(* Logix 5000 project; controller AMANA_DC_PLANT_01 vendor 1 type 14 code 164 rev 31.12; software revision 31.02; part 8 of 9 *)
(* tags used below, declared in another part *)
   Barcode_Longest : DINT;
   Barcode_Shortest : DINT;
   Comma : STRING;
   NULL_String : STRING;
   SCANNER_LN467MERGE_DATA : Keyence_2_Barcode;
   SCANNER_LONGTERMEAST_DATA : Keyence_2_Barcode;
   SCANNER_LONGTERMWEST_DATA : Keyence_2_Barcode;
   SCANNER_WAREHOUSENORTH_DATA : Keyence_2_Barcode;
   SCANNER_WAREHOUSESOUTH_DATA : Keyence_2_Barcode;
(* OH_BARCODE_SCAN, continued *)

ROUTINE R06_WAREHOUSENORTH   (* ladder *)
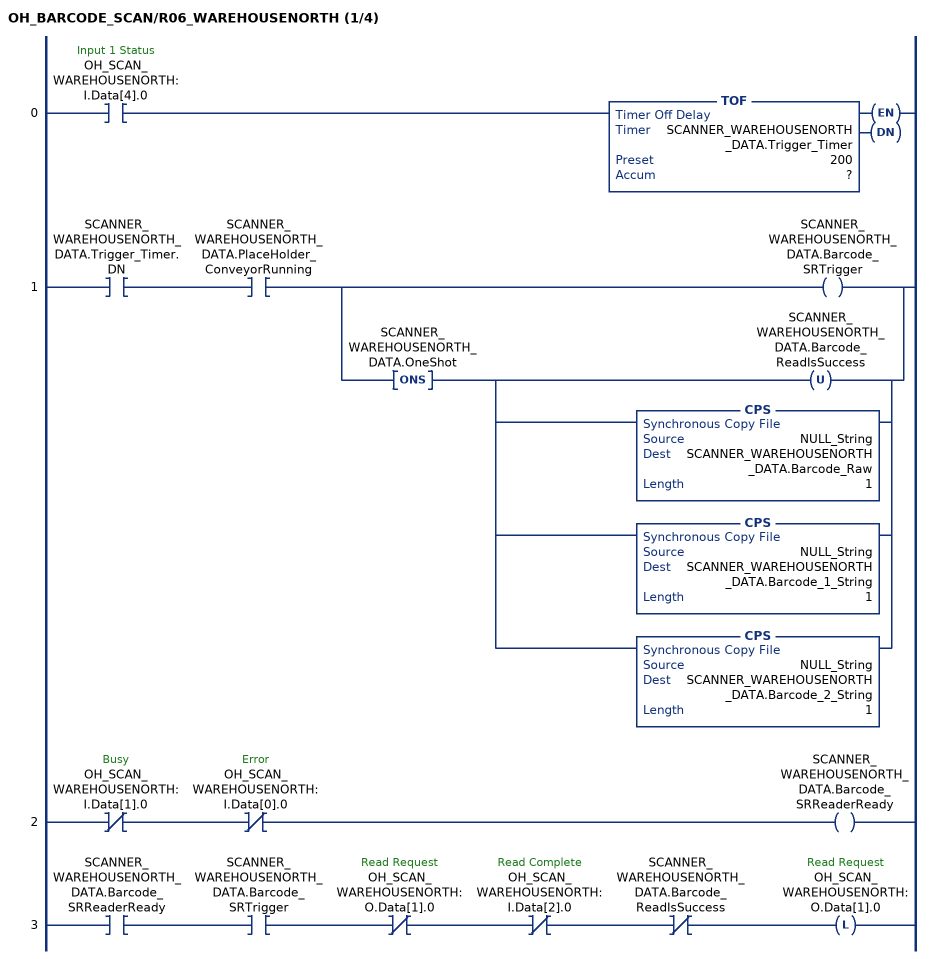
   0: XIC(OH_SCAN_WAREHOUSENORTH:I.Data[4].0)TOF(SCANNER_WAREHOUSENORTH_DATA.Trigger_Timer,?,?);
   1: XIC(SCANNER_WAREHOUSENORTH_DATA.Trigger_Timer.DN)XIC(SCANNER_WAREHOUSENORTH_DATA.PlaceHolder_ConveyorRunning)[OTE(SCANNER_WAREHOUSENORTH_DATA.Barcode_SRTrigger) ,ONS(SCANNER_WAREHOUSENORTH_DATA.OneShot) [OTU(SCANNER_WAREHOUSENORTH_DATA.Barcode_ReadIsSuccess) ,CPS(NULL_String,SCANNER_WAREHOUSENORTH_DATA.Barcode_Raw,1) ,CPS(NULL_String,SCANNER_WAREHOUSENORTH_DATA.Barcode_1_String,1) ,CPS(NULL_String,SCANNER_WAREHOUSENORTH_DATA.Barcode_2_String,1) ] ];
   2: XIO(OH_SCAN_WAREHOUSENORTH:I.Data[1].0)XIO(OH_SCAN_WAREHOUSENORTH:I.Data[0].0)OTE(SCANNER_WAREHOUSENORTH_DATA.Barcode_SRReaderReady);
   3: XIC(SCANNER_WAREHOUSENORTH_DATA.Barcode_SRReaderReady)XIC(SCANNER_WAREHOUSENORTH_DATA.Barcode_SRTrigger)XIO(OH_SCAN_WAREHOUSENORTH:O.Data[1].0)XIO(OH_SCAN_WAREHOUSENORTH:I.Data[2].0)XIO(SCANNER_WAREHOUSENORTH_DATA.Barcode_ReadIsSuccess)OTL(OH_SCAN_WAREHOUSENORTH:O.Data[1].0);
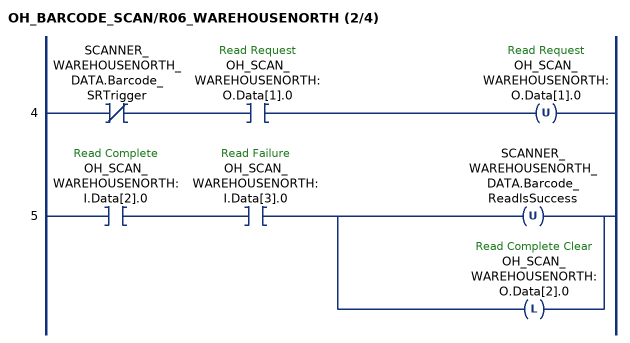
   4: XIO(SCANNER_WAREHOUSENORTH_DATA.Barcode_SRTrigger)XIC(OH_SCAN_WAREHOUSENORTH:O.Data[1].0)OTU(OH_SCAN_WAREHOUSENORTH:O.Data[1].0);
   5: XIC(OH_SCAN_WAREHOUSENORTH:I.Data[2].0)XIC(OH_SCAN_WAREHOUSENORTH:I.Data[3].0)[OTU(SCANNER_WAREHOUSENORTH_DATA.Barcode_ReadIsSuccess) ,OTL(OH_SCAN_WAREHOUSENORTH:O.Data[2].0) ];
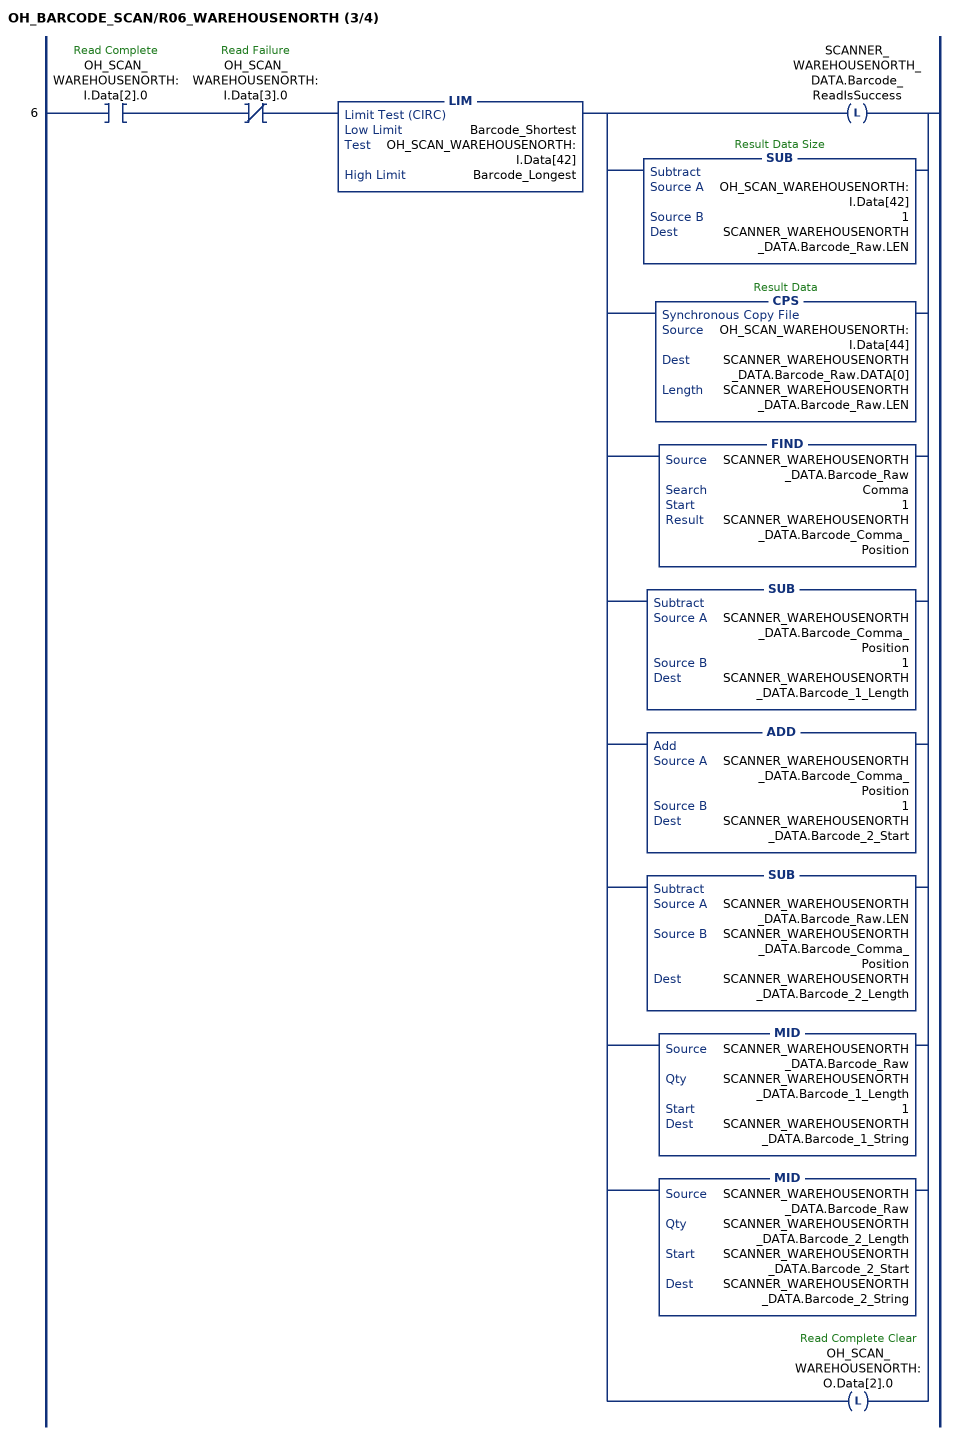
   6: XIC(OH_SCAN_WAREHOUSENORTH:I.Data[2].0)XIO(OH_SCAN_WAREHOUSENORTH:I.Data[3].0)LIM(Barcode_Shortest,OH_SCAN_WAREHOUSENORTH:I.Data[42],Barcode_Longest)[OTL(SCANNER_WAREHOUSENORTH_DATA.Barcode_ReadIsSuccess) ,SUB(OH_SCAN_WAREHOUSENORTH:I.Data[42],1,SCANNER_WAREHOUSENORTH_DATA.Barcode_Raw.LEN) ,CPS(OH_SCAN_WAREHOUSENORTH:I.Data[44],SCANNER_WAREHOUSENORTH_DATA.Barcode_Raw.DATA[0],SCANNER_WAREHOUSENORTH_DATA.Barcode_Raw.LEN) ,FIND(SCANNER_WAREHOUSENORTH_DATA.Barcode_Raw,Comma,1,SCANNER_WAREHOUSENORTH_DATA.Barcode_Comma_Position) ,SUB(SCANNER_WAREHOUSENORTH_DATA.Barcode_Comma_Position,1,SCANNER_WAREHOUSENORTH_DATA.Barcode_1_Length) ,ADD(SCANNER_WAREHOUSENORTH_DATA.Barcode_Comma_Position,1,SCANNER_WAREHOUSENORTH_DATA.Barcode_2_Start) ,SUB(SCANNER_WAREHOUSENORTH_DATA.Barcode_Raw.LEN,SCANNER_WAREHOUSENORTH_DATA.Barcode_Comma_Position,SCANNER_WAREHOUSENORTH_DATA.Barcode_2_Length) ,MID(SCANNER_WAREHOUSENORTH_DATA.Barcode_Raw,SCANNER_WAREHOUSENORTH_DATA.Barcode_1_Length,1,SCANNER_WAREHOUSENORTH_DATA.Barcode_1_String) ,MID(SCANNER_WAREHOUSENORTH_DATA.Barcode_Raw,SCANNER_WAREHOUSENORTH_DATA.Barcode_2_Length,SCANNER_WAREHOUSENORTH_DATA.Barcode_2_Start,SCANNER_WAREHOUSENORTH_DATA.Barcode_2_String) ,OTL(OH_SCAN_WAREHOUSENORTH:O.Data[2].0) ];
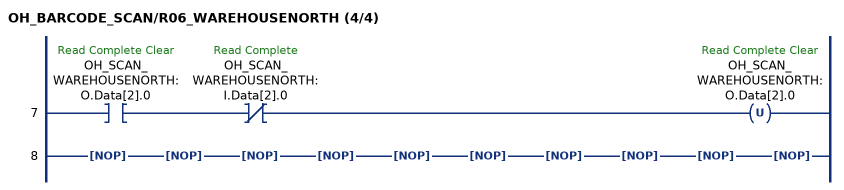
   7: XIC(OH_SCAN_WAREHOUSENORTH:O.Data[2].0)XIO(OH_SCAN_WAREHOUSENORTH:I.Data[2].0)OTU(OH_SCAN_WAREHOUSENORTH:O.Data[2].0);
   8: NOP()NOP()NOP()NOP()NOP()NOP()NOP()NOP()NOP()NOP();
END_ROUTINE

ROUTINE R07_WAREHOUSESOUTH   (* ladder *)
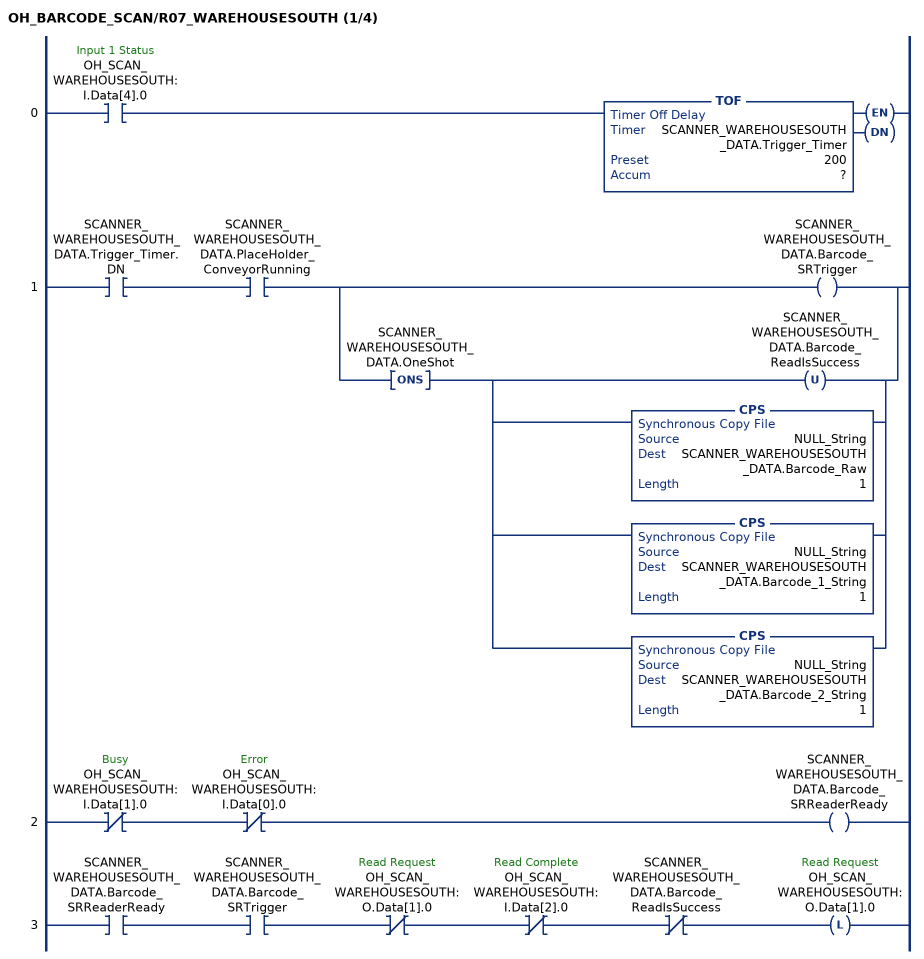
   0: XIC(OH_SCAN_WAREHOUSESOUTH:I.Data[4].0)TOF(SCANNER_WAREHOUSESOUTH_DATA.Trigger_Timer,?,?);
   1: XIC(SCANNER_WAREHOUSESOUTH_DATA.Trigger_Timer.DN)XIC(SCANNER_WAREHOUSESOUTH_DATA.PlaceHolder_ConveyorRunning)[OTE(SCANNER_WAREHOUSESOUTH_DATA.Barcode_SRTrigger) ,ONS(SCANNER_WAREHOUSESOUTH_DATA.OneShot) [OTU(SCANNER_WAREHOUSESOUTH_DATA.Barcode_ReadIsSuccess) ,CPS(NULL_String,SCANNER_WAREHOUSESOUTH_DATA.Barcode_Raw,1) ,CPS(NULL_String,SCANNER_WAREHOUSESOUTH_DATA.Barcode_1_String,1) ,CPS(NULL_String,SCANNER_WAREHOUSESOUTH_DATA.Barcode_2_String,1) ] ];
   2: XIO(OH_SCAN_WAREHOUSESOUTH:I.Data[1].0)XIO(OH_SCAN_WAREHOUSESOUTH:I.Data[0].0)OTE(SCANNER_WAREHOUSESOUTH_DATA.Barcode_SRReaderReady);
   3: XIC(SCANNER_WAREHOUSESOUTH_DATA.Barcode_SRReaderReady)XIC(SCANNER_WAREHOUSESOUTH_DATA.Barcode_SRTrigger)XIO(OH_SCAN_WAREHOUSESOUTH:O.Data[1].0)XIO(OH_SCAN_WAREHOUSESOUTH:I.Data[2].0)XIO(SCANNER_WAREHOUSESOUTH_DATA.Barcode_ReadIsSuccess)OTL(OH_SCAN_WAREHOUSESOUTH:O.Data[1].0);
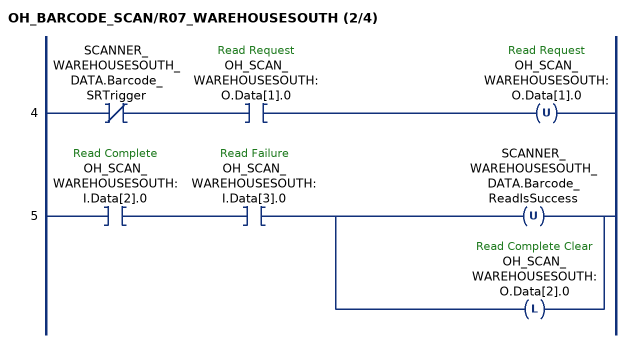
   4: XIO(SCANNER_WAREHOUSESOUTH_DATA.Barcode_SRTrigger)XIC(OH_SCAN_WAREHOUSESOUTH:O.Data[1].0)OTU(OH_SCAN_WAREHOUSESOUTH:O.Data[1].0);
   5: XIC(OH_SCAN_WAREHOUSESOUTH:I.Data[2].0)XIC(OH_SCAN_WAREHOUSESOUTH:I.Data[3].0)[OTU(SCANNER_WAREHOUSESOUTH_DATA.Barcode_ReadIsSuccess) ,OTL(OH_SCAN_WAREHOUSESOUTH:O.Data[2].0) ];
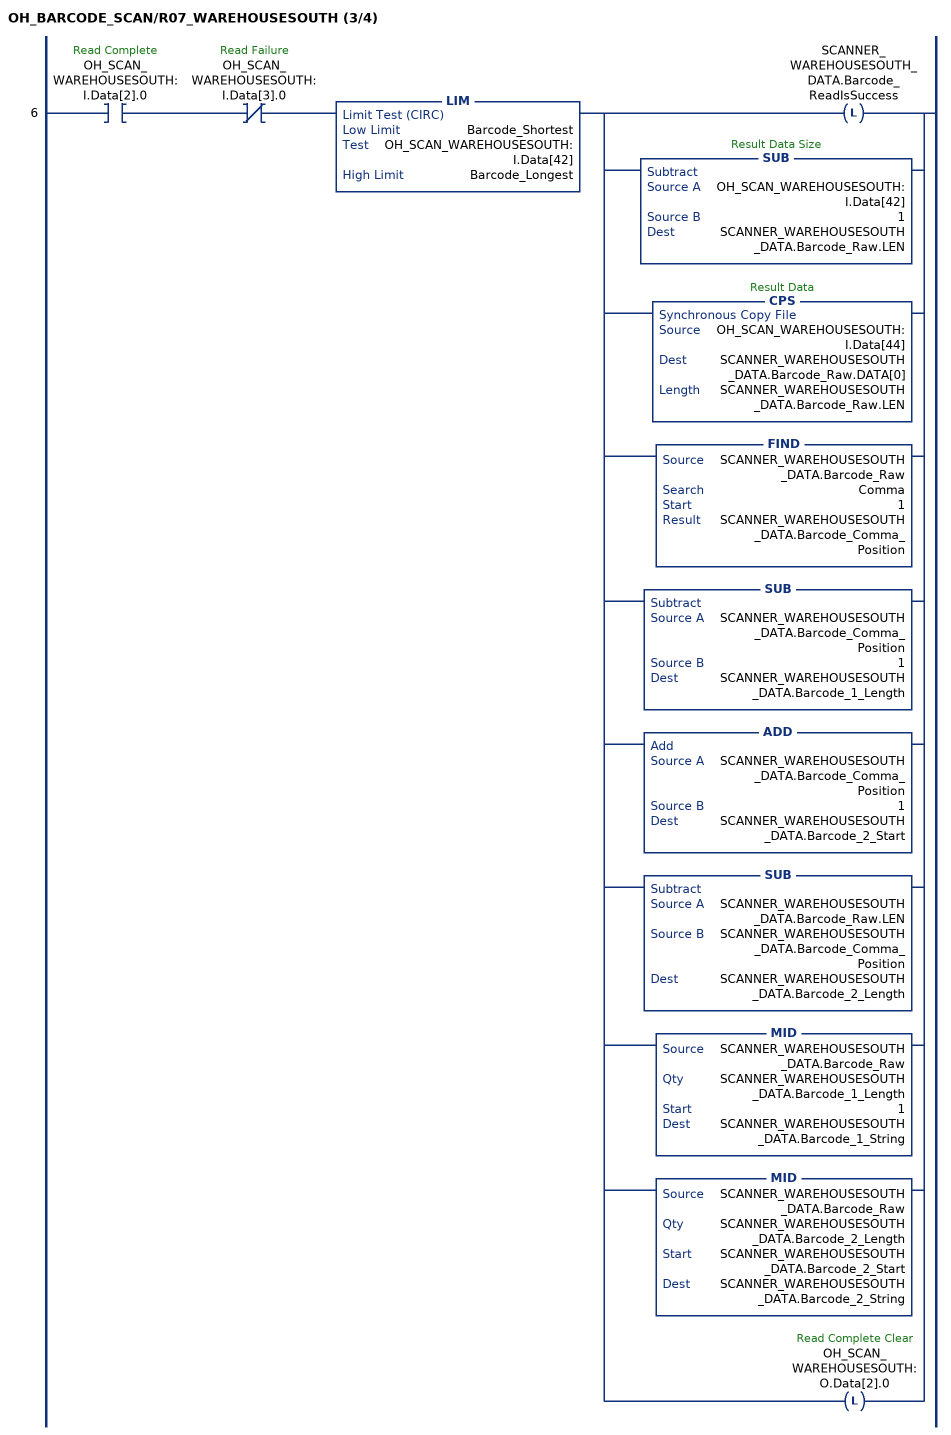
   6: XIC(OH_SCAN_WAREHOUSESOUTH:I.Data[2].0)XIO(OH_SCAN_WAREHOUSESOUTH:I.Data[3].0)LIM(Barcode_Shortest,OH_SCAN_WAREHOUSESOUTH:I.Data[42],Barcode_Longest)[OTL(SCANNER_WAREHOUSESOUTH_DATA.Barcode_ReadIsSuccess) ,SUB(OH_SCAN_WAREHOUSESOUTH:I.Data[42],1,SCANNER_WAREHOUSESOUTH_DATA.Barcode_Raw.LEN) ,CPS(OH_SCAN_WAREHOUSESOUTH:I.Data[44],SCANNER_WAREHOUSESOUTH_DATA.Barcode_Raw.DATA[0],SCANNER_WAREHOUSESOUTH_DATA.Barcode_Raw.LEN) ,FIND(SCANNER_WAREHOUSESOUTH_DATA.Barcode_Raw,Comma,1,SCANNER_WAREHOUSESOUTH_DATA.Barcode_Comma_Position) ,SUB(SCANNER_WAREHOUSESOUTH_DATA.Barcode_Comma_Position,1,SCANNER_WAREHOUSESOUTH_DATA.Barcode_1_Length) ,ADD(SCANNER_WAREHOUSESOUTH_DATA.Barcode_Comma_Position,1,SCANNER_WAREHOUSESOUTH_DATA.Barcode_2_Start) ,SUB(SCANNER_WAREHOUSESOUTH_DATA.Barcode_Raw.LEN,SCANNER_WAREHOUSESOUTH_DATA.Barcode_Comma_Position,SCANNER_WAREHOUSESOUTH_DATA.Barcode_2_Length) ,MID(SCANNER_WAREHOUSESOUTH_DATA.Barcode_Raw,SCANNER_WAREHOUSESOUTH_DATA.Barcode_1_Length,1,SCANNER_WAREHOUSESOUTH_DATA.Barcode_1_String) ,MID(SCANNER_WAREHOUSESOUTH_DATA.Barcode_Raw,SCANNER_WAREHOUSESOUTH_DATA.Barcode_2_Length,SCANNER_WAREHOUSESOUTH_DATA.Barcode_2_Start,SCANNER_WAREHOUSESOUTH_DATA.Barcode_2_String) ,OTL(OH_SCAN_WAREHOUSESOUTH:O.Data[2].0) ];
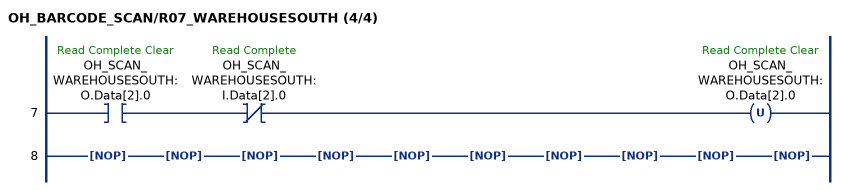
   7: XIC(OH_SCAN_WAREHOUSESOUTH:O.Data[2].0)XIO(OH_SCAN_WAREHOUSESOUTH:I.Data[2].0)OTU(OH_SCAN_WAREHOUSESOUTH:O.Data[2].0);
   8: NOP()NOP()NOP()NOP()NOP()NOP()NOP()NOP()NOP()NOP();
END_ROUTINE

ROUTINE R08_LONGTERMEAST   (* ladder *)
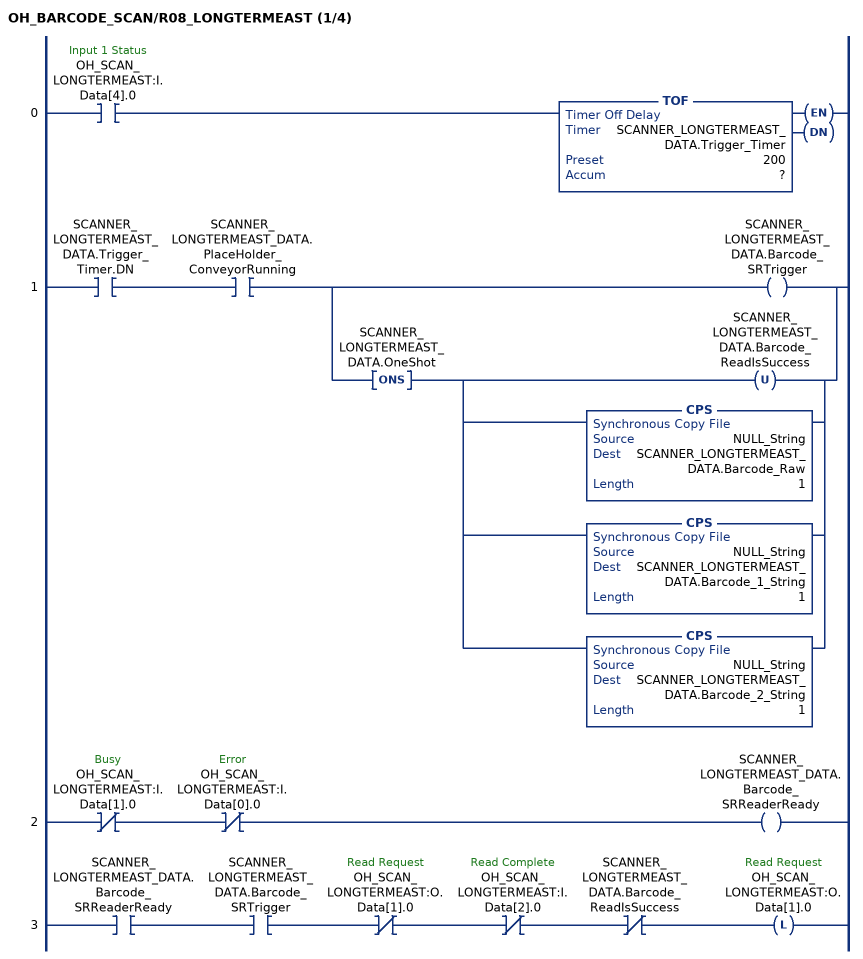
   0: XIC(OH_SCAN_LONGTERMEAST:I.Data[4].0)TOF(SCANNER_LONGTERMEAST_DATA.Trigger_Timer,?,?);
   1: XIC(SCANNER_LONGTERMEAST_DATA.Trigger_Timer.DN)XIC(SCANNER_LONGTERMEAST_DATA.PlaceHolder_ConveyorRunning)[OTE(SCANNER_LONGTERMEAST_DATA.Barcode_SRTrigger) ,ONS(SCANNER_LONGTERMEAST_DATA.OneShot) [OTU(SCANNER_LONGTERMEAST_DATA.Barcode_ReadIsSuccess) ,CPS(NULL_String,SCANNER_LONGTERMEAST_DATA.Barcode_Raw,1) ,CPS(NULL_String,SCANNER_LONGTERMEAST_DATA.Barcode_1_String,1) ,CPS(NULL_String,SCANNER_LONGTERMEAST_DATA.Barcode_2_String,1) ] ];
   2: XIO(OH_SCAN_LONGTERMEAST:I.Data[1].0)XIO(OH_SCAN_LONGTERMEAST:I.Data[0].0)OTE(SCANNER_LONGTERMEAST_DATA.Barcode_SRReaderReady);
   3: XIC(SCANNER_LONGTERMEAST_DATA.Barcode_SRReaderReady)XIC(SCANNER_LONGTERMEAST_DATA.Barcode_SRTrigger)XIO(OH_SCAN_LONGTERMEAST:O.Data[1].0)XIO(OH_SCAN_LONGTERMEAST:I.Data[2].0)XIO(SCANNER_LONGTERMEAST_DATA.Barcode_ReadIsSuccess)OTL(OH_SCAN_LONGTERMEAST:O.Data[1].0);
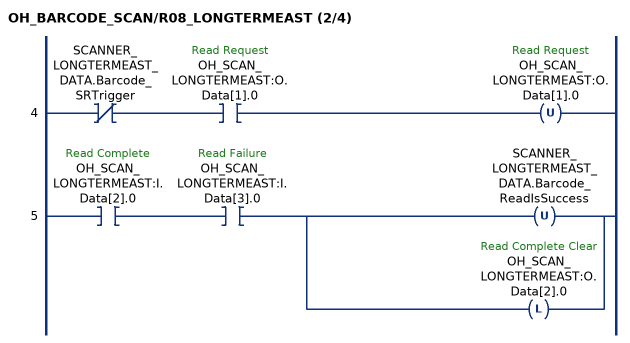
   4: XIO(SCANNER_LONGTERMEAST_DATA.Barcode_SRTrigger)XIC(OH_SCAN_LONGTERMEAST:O.Data[1].0)OTU(OH_SCAN_LONGTERMEAST:O.Data[1].0);
   5: XIC(OH_SCAN_LONGTERMEAST:I.Data[2].0)XIC(OH_SCAN_LONGTERMEAST:I.Data[3].0)[OTU(SCANNER_LONGTERMEAST_DATA.Barcode_ReadIsSuccess) ,OTL(OH_SCAN_LONGTERMEAST:O.Data[2].0) ];
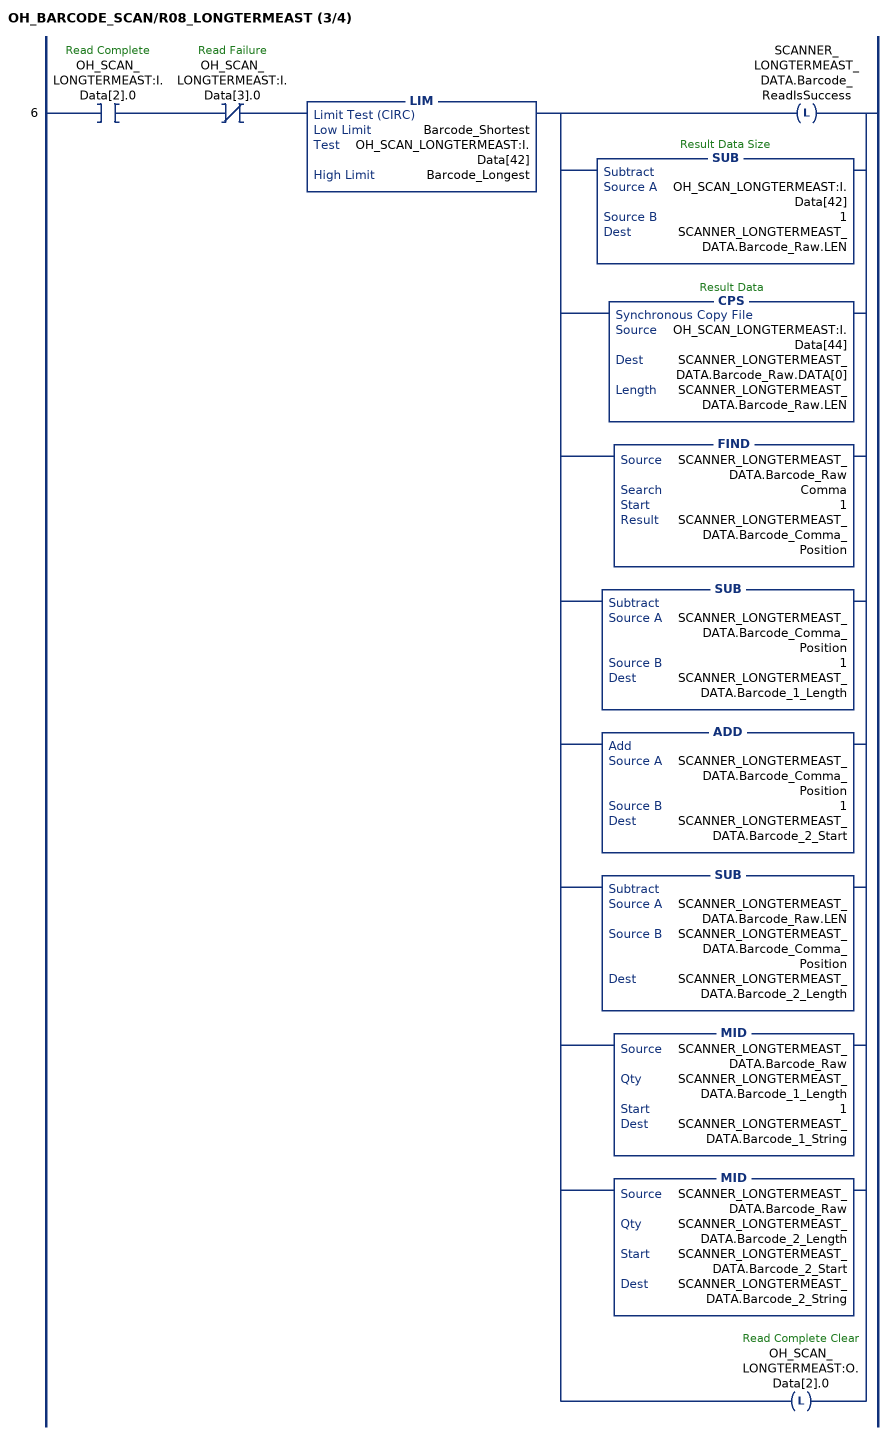
   6: XIC(OH_SCAN_LONGTERMEAST:I.Data[2].0)XIO(OH_SCAN_LONGTERMEAST:I.Data[3].0)LIM(Barcode_Shortest,OH_SCAN_LONGTERMEAST:I.Data[42],Barcode_Longest)[OTL(SCANNER_LONGTERMEAST_DATA.Barcode_ReadIsSuccess) ,SUB(OH_SCAN_LONGTERMEAST:I.Data[42],1,SCANNER_LONGTERMEAST_DATA.Barcode_Raw.LEN) ,CPS(OH_SCAN_LONGTERMEAST:I.Data[44],SCANNER_LONGTERMEAST_DATA.Barcode_Raw.DATA[0],SCANNER_LONGTERMEAST_DATA.Barcode_Raw.LEN) ,FIND(SCANNER_LONGTERMEAST_DATA.Barcode_Raw,Comma,1,SCANNER_LONGTERMEAST_DATA.Barcode_Comma_Position) ,SUB(SCANNER_LONGTERMEAST_DATA.Barcode_Comma_Position,1,SCANNER_LONGTERMEAST_DATA.Barcode_1_Length) ,ADD(SCANNER_LONGTERMEAST_DATA.Barcode_Comma_Position,1,SCANNER_LONGTERMEAST_DATA.Barcode_2_Start) ,SUB(SCANNER_LONGTERMEAST_DATA.Barcode_Raw.LEN,SCANNER_LONGTERMEAST_DATA.Barcode_Comma_Position,SCANNER_LONGTERMEAST_DATA.Barcode_2_Length) ,MID(SCANNER_LONGTERMEAST_DATA.Barcode_Raw,SCANNER_LONGTERMEAST_DATA.Barcode_1_Length,1,SCANNER_LONGTERMEAST_DATA.Barcode_1_String) ,MID(SCANNER_LONGTERMEAST_DATA.Barcode_Raw,SCANNER_LONGTERMEAST_DATA.Barcode_2_Length,SCANNER_LONGTERMEAST_DATA.Barcode_2_Start,SCANNER_LONGTERMEAST_DATA.Barcode_2_String) ,OTL(OH_SCAN_LONGTERMEAST:O.Data[2].0) ];
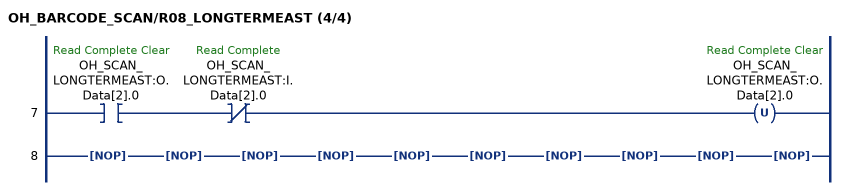
   7: XIC(OH_SCAN_LONGTERMEAST:O.Data[2].0)XIO(OH_SCAN_LONGTERMEAST:I.Data[2].0)OTU(OH_SCAN_LONGTERMEAST:O.Data[2].0);
   8: NOP()NOP()NOP()NOP()NOP()NOP()NOP()NOP()NOP()NOP();
END_ROUTINE

ROUTINE R09_LONGTERMWEST   (* ladder *)
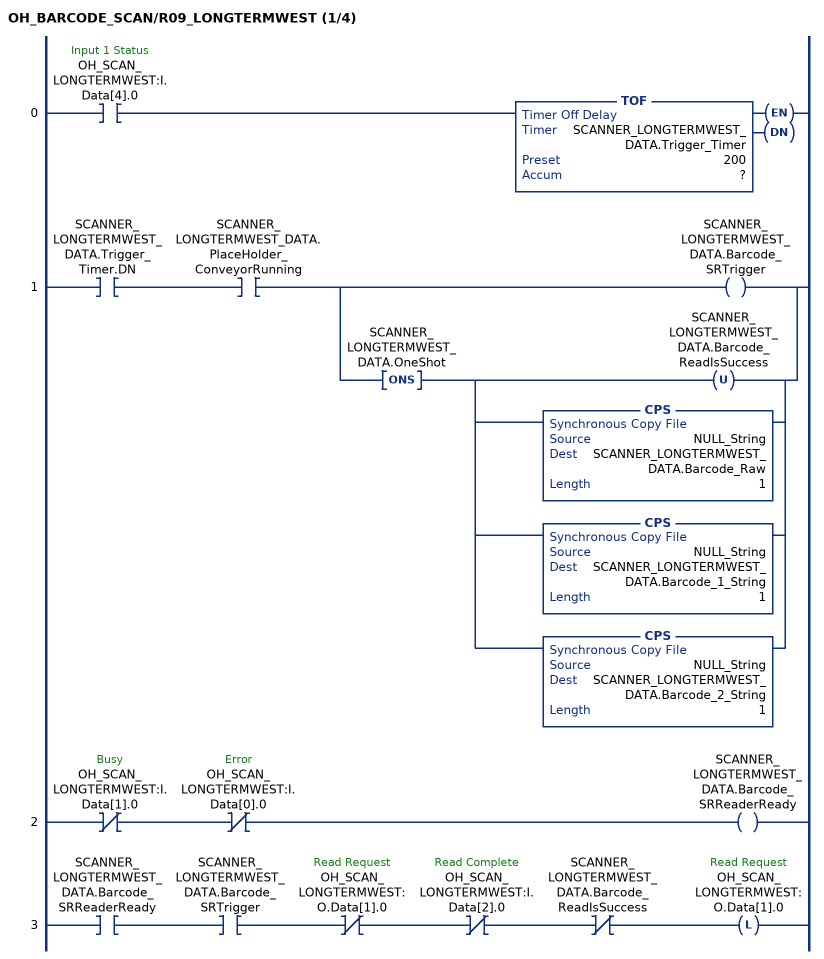
   0: XIC(OH_SCAN_LONGTERMWEST:I.Data[4].0)TOF(SCANNER_LONGTERMWEST_DATA.Trigger_Timer,?,?);
   1: XIC(SCANNER_LONGTERMWEST_DATA.Trigger_Timer.DN)XIC(SCANNER_LONGTERMWEST_DATA.PlaceHolder_ConveyorRunning)[OTE(SCANNER_LONGTERMWEST_DATA.Barcode_SRTrigger) ,ONS(SCANNER_LONGTERMWEST_DATA.OneShot) [OTU(SCANNER_LONGTERMWEST_DATA.Barcode_ReadIsSuccess) ,CPS(NULL_String,SCANNER_LONGTERMWEST_DATA.Barcode_Raw,1) ,CPS(NULL_String,SCANNER_LONGTERMWEST_DATA.Barcode_1_String,1) ,CPS(NULL_String,SCANNER_LONGTERMWEST_DATA.Barcode_2_String,1) ] ];
   2: XIO(OH_SCAN_LONGTERMWEST:I.Data[1].0)XIO(OH_SCAN_LONGTERMWEST:I.Data[0].0)OTE(SCANNER_LONGTERMWEST_DATA.Barcode_SRReaderReady);
   3: XIC(SCANNER_LONGTERMWEST_DATA.Barcode_SRReaderReady)XIC(SCANNER_LONGTERMWEST_DATA.Barcode_SRTrigger)XIO(OH_SCAN_LONGTERMWEST:O.Data[1].0)XIO(OH_SCAN_LONGTERMWEST:I.Data[2].0)XIO(SCANNER_LONGTERMWEST_DATA.Barcode_ReadIsSuccess)OTL(OH_SCAN_LONGTERMWEST:O.Data[1].0);
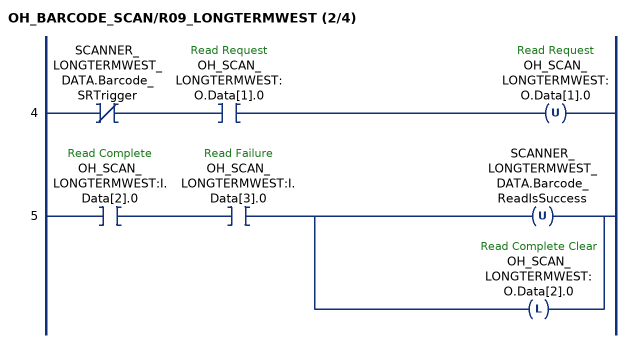
   4: XIO(SCANNER_LONGTERMWEST_DATA.Barcode_SRTrigger)XIC(OH_SCAN_LONGTERMWEST:O.Data[1].0)OTU(OH_SCAN_LONGTERMWEST:O.Data[1].0);
   5: XIC(OH_SCAN_LONGTERMWEST:I.Data[2].0)XIC(OH_SCAN_LONGTERMWEST:I.Data[3].0)[OTU(SCANNER_LONGTERMWEST_DATA.Barcode_ReadIsSuccess) ,OTL(OH_SCAN_LONGTERMWEST:O.Data[2].0) ];
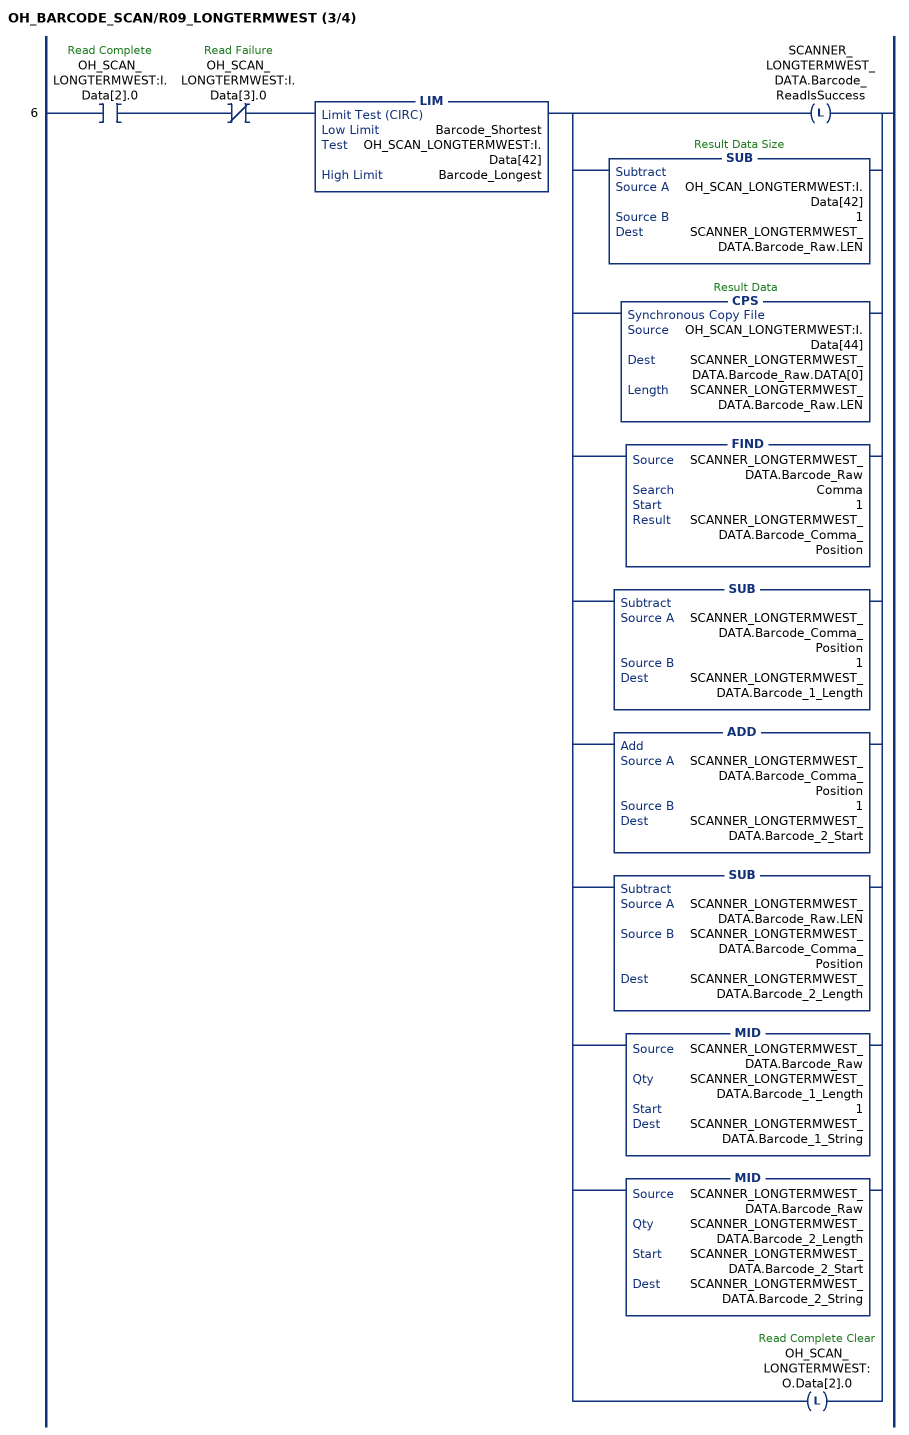
   6: XIC(OH_SCAN_LONGTERMWEST:I.Data[2].0)XIO(OH_SCAN_LONGTERMWEST:I.Data[3].0)LIM(Barcode_Shortest,OH_SCAN_LONGTERMWEST:I.Data[42],Barcode_Longest)[OTL(SCANNER_LONGTERMWEST_DATA.Barcode_ReadIsSuccess) ,SUB(OH_SCAN_LONGTERMWEST:I.Data[42],1,SCANNER_LONGTERMWEST_DATA.Barcode_Raw.LEN) ,CPS(OH_SCAN_LONGTERMWEST:I.Data[44],SCANNER_LONGTERMWEST_DATA.Barcode_Raw.DATA[0],SCANNER_LONGTERMWEST_DATA.Barcode_Raw.LEN) ,FIND(SCANNER_LONGTERMWEST_DATA.Barcode_Raw,Comma,1,SCANNER_LONGTERMWEST_DATA.Barcode_Comma_Position) ,SUB(SCANNER_LONGTERMWEST_DATA.Barcode_Comma_Position,1,SCANNER_LONGTERMWEST_DATA.Barcode_1_Length) ,ADD(SCANNER_LONGTERMWEST_DATA.Barcode_Comma_Position,1,SCANNER_LONGTERMWEST_DATA.Barcode_2_Start) ,SUB(SCANNER_LONGTERMWEST_DATA.Barcode_Raw.LEN,SCANNER_LONGTERMWEST_DATA.Barcode_Comma_Position,SCANNER_LONGTERMWEST_DATA.Barcode_2_Length) ,MID(SCANNER_LONGTERMWEST_DATA.Barcode_Raw,SCANNER_LONGTERMWEST_DATA.Barcode_1_Length,1,SCANNER_LONGTERMWEST_DATA.Barcode_1_String) ,MID(SCANNER_LONGTERMWEST_DATA.Barcode_Raw,SCANNER_LONGTERMWEST_DATA.Barcode_2_Length,SCANNER_LONGTERMWEST_DATA.Barcode_2_Start,SCANNER_LONGTERMWEST_DATA.Barcode_2_String) ,OTL(OH_SCAN_LONGTERMWEST:O.Data[2].0) ];
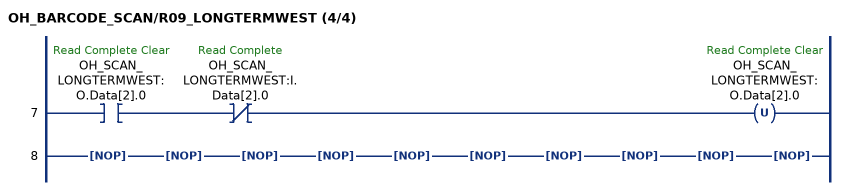
   7: XIC(OH_SCAN_LONGTERMWEST:O.Data[2].0)XIO(OH_SCAN_LONGTERMWEST:I.Data[2].0)OTU(OH_SCAN_LONGTERMWEST:O.Data[2].0);
   8: NOP()NOP()NOP()NOP()NOP()NOP()NOP()NOP()NOP()NOP();
END_ROUTINE

ROUTINE R10_LN467MERGE   (* ladder *)
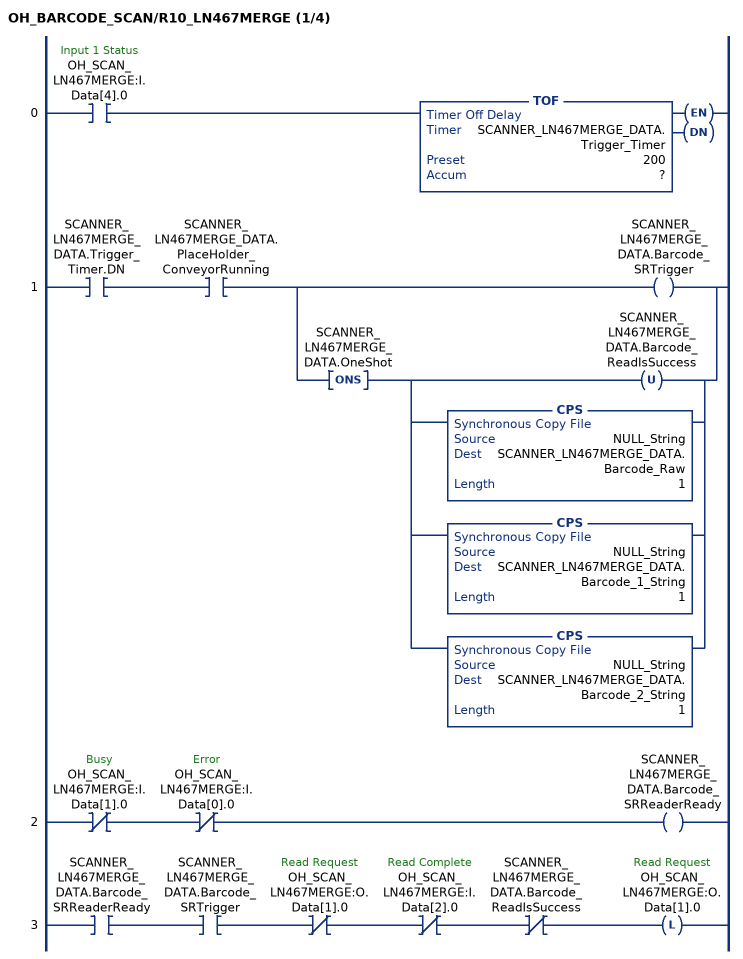
   0: XIC(OH_SCAN_LN467MERGE:I.Data[4].0)TOF(SCANNER_LN467MERGE_DATA.Trigger_Timer,?,?);
   1: XIC(SCANNER_LN467MERGE_DATA.Trigger_Timer.DN)XIC(SCANNER_LN467MERGE_DATA.PlaceHolder_ConveyorRunning)[OTE(SCANNER_LN467MERGE_DATA.Barcode_SRTrigger) ,ONS(SCANNER_LN467MERGE_DATA.OneShot) [OTU(SCANNER_LN467MERGE_DATA.Barcode_ReadIsSuccess) ,CPS(NULL_String,SCANNER_LN467MERGE_DATA.Barcode_Raw,1) ,CPS(NULL_String,SCANNER_LN467MERGE_DATA.Barcode_1_String,1) ,CPS(NULL_String,SCANNER_LN467MERGE_DATA.Barcode_2_String,1) ] ];
   2: XIO(OH_SCAN_LN467MERGE:I.Data[1].0)XIO(OH_SCAN_LN467MERGE:I.Data[0].0)OTE(SCANNER_LN467MERGE_DATA.Barcode_SRReaderReady);
   3: XIC(SCANNER_LN467MERGE_DATA.Barcode_SRReaderReady)XIC(SCANNER_LN467MERGE_DATA.Barcode_SRTrigger)XIO(OH_SCAN_LN467MERGE:O.Data[1].0)XIO(OH_SCAN_LN467MERGE:I.Data[2].0)XIO(SCANNER_LN467MERGE_DATA.Barcode_ReadIsSuccess)OTL(OH_SCAN_LN467MERGE:O.Data[1].0);
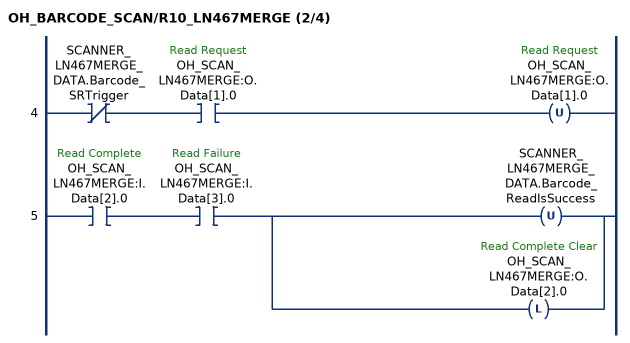
   4: XIO(SCANNER_LN467MERGE_DATA.Barcode_SRTrigger)XIC(OH_SCAN_LN467MERGE:O.Data[1].0)OTU(OH_SCAN_LN467MERGE:O.Data[1].0);
   5: XIC(OH_SCAN_LN467MERGE:I.Data[2].0)XIC(OH_SCAN_LN467MERGE:I.Data[3].0)[OTU(SCANNER_LN467MERGE_DATA.Barcode_ReadIsSuccess) ,OTL(OH_SCAN_LN467MERGE:O.Data[2].0) ];
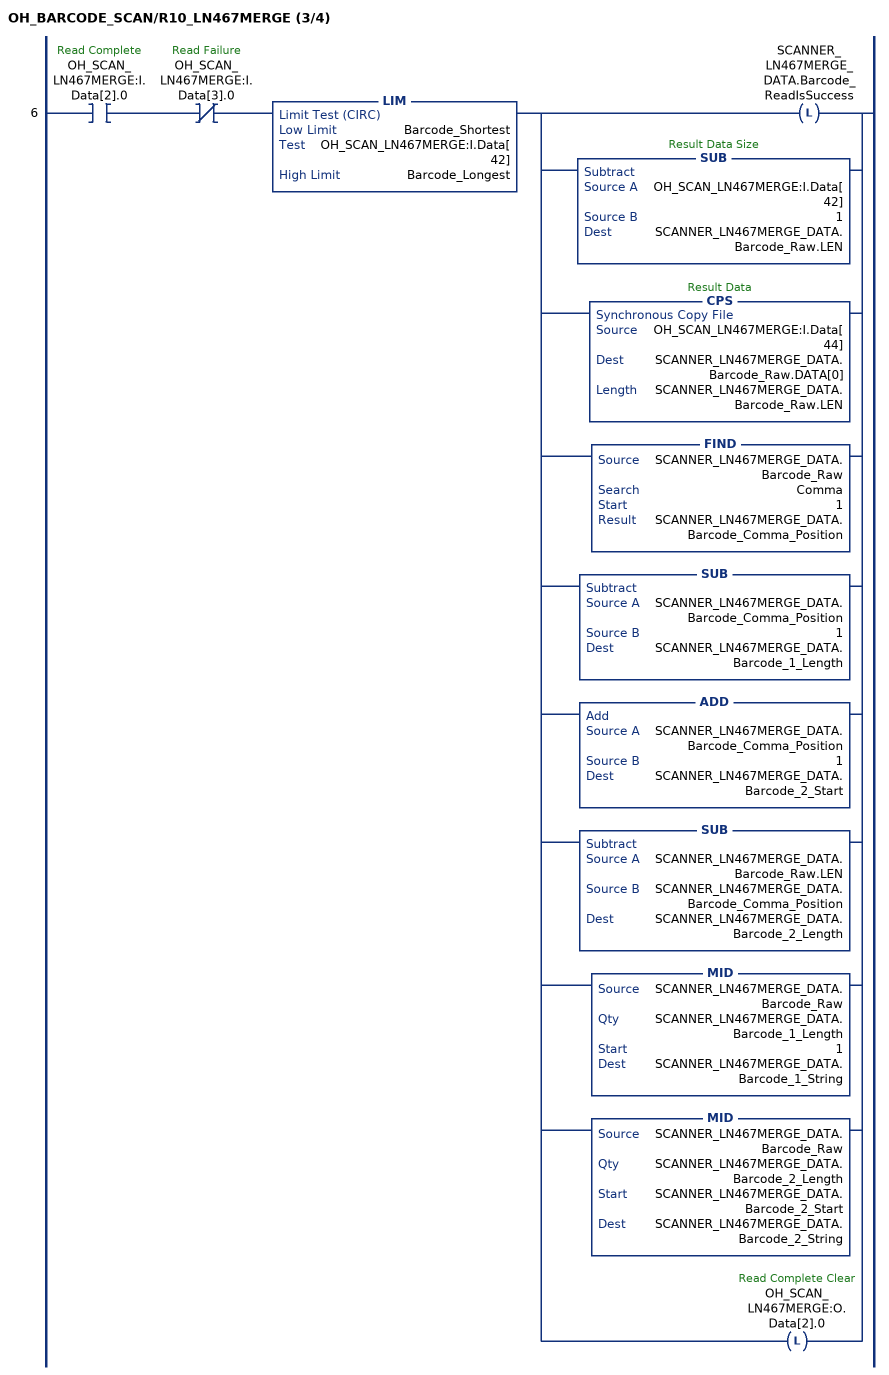
   6: XIC(OH_SCAN_LN467MERGE:I.Data[2].0)XIO(OH_SCAN_LN467MERGE:I.Data[3].0)LIM(Barcode_Shortest,OH_SCAN_LN467MERGE:I.Data[42],Barcode_Longest)[OTL(SCANNER_LN467MERGE_DATA.Barcode_ReadIsSuccess) ,SUB(OH_SCAN_LN467MERGE:I.Data[42],1,SCANNER_LN467MERGE_DATA.Barcode_Raw.LEN) ,CPS(OH_SCAN_LN467MERGE:I.Data[44],SCANNER_LN467MERGE_DATA.Barcode_Raw.DATA[0],SCANNER_LN467MERGE_DATA.Barcode_Raw.LEN) ,FIND(SCANNER_LN467MERGE_DATA.Barcode_Raw,Comma,1,SCANNER_LN467MERGE_DATA.Barcode_Comma_Position) ,SUB(SCANNER_LN467MERGE_DATA.Barcode_Comma_Position,1,SCANNER_LN467MERGE_DATA.Barcode_1_Length) ,ADD(SCANNER_LN467MERGE_DATA.Barcode_Comma_Position,1,SCANNER_LN467MERGE_DATA.Barcode_2_Start) ,SUB(SCANNER_LN467MERGE_DATA.Barcode_Raw.LEN,SCANNER_LN467MERGE_DATA.Barcode_Comma_Position,SCANNER_LN467MERGE_DATA.Barcode_2_Length) ,MID(SCANNER_LN467MERGE_DATA.Barcode_Raw,SCANNER_LN467MERGE_DATA.Barcode_1_Length,1,SCANNER_LN467MERGE_DATA.Barcode_1_String) ,MID(SCANNER_LN467MERGE_DATA.Barcode_Raw,SCANNER_LN467MERGE_DATA.Barcode_2_Length,SCANNER_LN467MERGE_DATA.Barcode_2_Start,SCANNER_LN467MERGE_DATA.Barcode_2_String) ,OTL(OH_SCAN_LN467MERGE:O.Data[2].0) ];
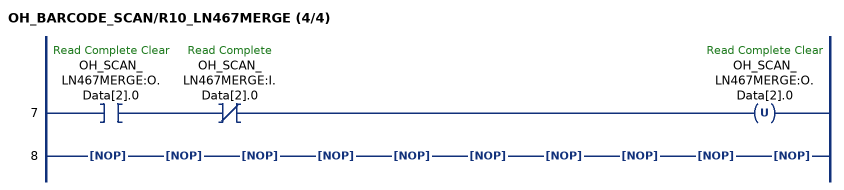
   7: XIC(OH_SCAN_LN467MERGE:O.Data[2].0)XIO(OH_SCAN_LN467MERGE:I.Data[2].0)OTU(OH_SCAN_LN467MERGE:O.Data[2].0);
   8: NOP()NOP()NOP()NOP()NOP()NOP()NOP()NOP()NOP()NOP();
END_ROUTINE
